(*
SPDX-FileCopyrightText: © 2026 Oleksandr Tiutyk <trofimich@gmail.com>
SPDX-License-Identifier: MIT
License: https://opensource.org/license/mit
*)

(*!
<summary>Exchanges commands and status between an HMI and an automation component.</summary>
<description>
Derived elements supply component identity and invoke the protected update methods. Error timestamps are reset
to the epoch when no error is reported. Commands received in AutomationComponentCommands are consumed and reset
within the element instance upon dispatch. External HMI systems must write directly to the element's
AutomationComponentCommands symbol or read back the reset state for command handshake.
</description>
*)

FUNCTION_BLOCK ABSTRACT HmiAutomationComponentElement
VAR_INPUT
	AutomationComponentCommands : HMI_AUTOMATION_COMPONENT_COMMANDS;
END_VAR
VAR_OUTPUT
	AutomationComponentStatuses : HMI_AUTOMATION_COMPONENT_STATUSES;
END_VAR

(*!
<summary>Gets the class name of the concrete HMI element.</summary>
*)
{attribute 'monitoring' := 'call'}
PROPERTY ABSTRACT ClassName : REFERENCE TO STRING
GET
END_GET
END_PROPERTY

(*!
<summary>Gets the namespace of the concrete HMI element.</summary>
*)
{attribute 'monitoring' := 'call'}
PROPERTY ABSTRACT NamespaceName : REFERENCE TO STRING
GET
END_GET
END_PROPERTY

(*!
<summary>Dispatches pending HMI commands to the target automation component.</summary>
<description>
Captures and resets the command flags in AutomationComponentCommands to FALSE before invoking Enable,
Disable, or Reset on the target component, preventing repeated execution across cycles if a hook raises an
exception. When both Disable and Enable are set simultaneously, Disable takes precedence. A null component
reference causes an immediate return without mutating commands. External HMI systems must write directly to
the element's AutomationComponentCommands symbol or read back the reset state for command handshake.
</description>
<param name="automationComponent">Target component receiving the dispatched commands.</param>
*)
METHOD PROTECTED ProcessAutomationComponentCommands
VAR_INPUT
	automationComponent : IAutomationComponent;
END_VAR
VAR
	disableRequested : BOOL;
	enableRequested : BOOL;
	resetRequested : BOOL;
END_VAR
IF automationComponent = 0 THEN
	RETURN;
END_IF

disableRequested := AutomationComponentCommands.Disable;
enableRequested := AutomationComponentCommands.Enable;
resetRequested := AutomationComponentCommands.Reset;

AutomationComponentCommands.Disable := FALSE;
AutomationComponentCommands.Enable := FALSE;
AutomationComponentCommands.Reset := FALSE;

IF disableRequested THEN
	automationComponent.Disable();
ELSIF enableRequested THEN
	automationComponent.Enable(includeChildren := TRUE);
END_IF

IF resetRequested THEN
	automationComponent.Reset();
END_IF
END_METHOD

(*!
<summary>Copies current component status to the HMI outputs.</summary>
<description>
A null component leaves outputs unchanged. When no error is reported, clears error text and resets error
timestamps to LongDateAndTimes.EPOCH.
</description>
*)
METHOD PROTECTED UpdateAutomationComponentStatuses
VAR_INPUT
	automationComponent : IAutomationComponent;
END_VAR
IF automationComponent = 0 THEN
	RETURN;
END_IF

AutomationComponentStatuses.Enabled := automationComponent.Enabled;

AutomationComponentStatuses.HasError := automationComponent.HasError;

IF automationComponent.HasError THEN
	AutomationComponentStatuses.ErrorMessage := automationComponent.Error.ToString(
		sourceDisplayMode := TOF_Core.ERROR_SOURCE_DISPLAY_MODE.HIDDEN,
		timestampDisplayMode := TOF_Core.TIMESTAMP_DISPLAY_MODE.HIDDEN
	);
	AutomationComponentStatuses.ErrorSource := automationComponent.Error.GetSource(appendRootSource := TRUE);	
	AutomationComponentStatuses.ErrorLocalTimestamp := automationComponent.Error.LocalTimestamp;
	AutomationComponentStatuses.ErrorUtcTimestamp := automationComponent.Error.UtcTimestamp;
ELSE
	AutomationComponentStatuses.ErrorMessage := "";
	AutomationComponentStatuses.ErrorSource := '';	
	AutomationComponentStatuses.ErrorLocalTimestamp := TOF_Core.LongDateAndTimes.EPOCH;
	AutomationComponentStatuses.ErrorUtcTimestamp := TOF_Core.LongDateAndTimes.EPOCH;
END_IF

AutomationComponentStatuses.OperationalState := automationComponent.OperationalState;
AutomationComponentStatuses.OperationalStateName := TO_STRING(AutomationComponentStatuses.OperationalState);
AutomationComponentStatuses.OperationalStateReason := automationComponent.OperationalStateReason;
END_METHOD

END_FUNCTION_BLOCK

(* stored: Version 1.1.0.1
   POU HmiAutomationComponentElement: Id {dfcc69f0-a3dd-4c3d-a891-2d135d1b66d4}, SpecialFunc None
   Property ClassName: Id {68bc9c5e-2bbb-41cc-9f58-1693b2fff252}
   Get Get: Id {c765939a-c5a7-4ad9-9d08-f290090d46bf}
   Property NamespaceName: Id {bda4d4aa-e177-4633-8aad-fea890343f42}
   Get Get: Id {c9ed4c86-67cf-4c3c-ac55-ac69db7570aa}
   Method ProcessAutomationComponentCommands: Id {207422e4-4aeb-4d7d-a75d-782bbafe57cc}
   Method UpdateAutomationComponentStatuses: Id {7f185188-8a4b-421d-8d7b-e49d8614968d} *)
